PROGRAM MAIN
VAR
END_VAR

(* Application Engineer: LucasK *)
(* MQTT Sample to TecnoProcess Test *) 
(* Using Mosquitto MQTT Open Source Server *)
(* And MQTT-Explorer to test *)
(* start mosquitto with net start mosquitto *)

END_PROGRAM

(* stored: Version 1.1.0.1, ProductVersion 3.1.4024.12
   POU MAIN: Id {b8bf13c9-c2a9-42cb-95bd-2f6f16a1c3b2}, SpecialFunc None *)
